Yaskawa INFORM job: BUFFER_WAIT.JBI

/JOB
//NAME BUFFER_WAIT
//POS
///NPOS 0,0,0,0,0,0
//INST
///DATE 2011/11/29 21:45
///ATTR SC,RW
///GROUP1 RB1
NOP
WHILE I091>=I092
ENDWHILE
INC I091
END
